// TIA Portal project "Hydaulikaggregat" (V14)

(* hardware
DEVICE "S7-1200-Station_1"  S7-1200 Station
   slot 0: "Baugruppenträger_0"  Rack  V1.0
   slot 1: "PLC"  CPU 1214C DC/DC/DC  6ES7 214-1AG40-0XB0  V4.1
   slot 3: "AQ 1x12BIT_1"  6ES7 232-4HA30-0XB0  V1.0
DEVICE "HMI"  KTP700 Basic PN
   slot 0: "HMI"  HMI  6AV2 123-2GB03-0AX0  13.0.1.0
   slot 1: "HMI_RT_1"  KTP700 Basic PN  6AV2 123-2GB03-0AX0  13.0.1.0
   slot 5: "HMI.IE_CP_1"  PROFINET Schnittstelle
      slot 1: "PROFINET Schnittstelle_1"  PROFINET Schnittstelle
         slot 1: "Port_1"  Port
*)

// ===== PLC "PLC"  CPU 1214C DC/DC/DC =====

VAR_GLOBAL   // PLC tag table "Standard-Variablentabelle"
   "System_Byte" AT %MB100 : Byte;
   "FirstScan" AT %M100.0 : Bool;
   "DiagStatusUpdate" AT %M100.1 : Bool;
   "AlwaysTRUE" AT %M100.2 : Bool;
   "AlwaysFALSE" AT %M100.3 : Bool;
   "Clock_Byte" AT %MB110 : Byte;
   "Clock_10Hz" AT %M110.0 : Bool;
   "Clock_5Hz" AT %M110.1 : Bool;
   "Clock_2.5Hz" AT %M110.2 : Bool;
   "Clock_2Hz" AT %M110.3 : Bool;
   "Clock_1.25Hz" AT %M110.4 : Bool;
   "Clock_1Hz" AT %M110.5 : Bool;
   "Clock_0.625Hz" AT %M110.6 : Bool;
   "Clock_0.5Hz" AT %M110.7 : Bool;
   "S1 Taster Start" AT %Q0.0 : Bool;
   "S2 Taster Stop" AT %Q0.1 : Bool;
   "S3 Taster Quittieren" AT %Q0.2 : Bool;
   "B1Füllstand Ölbehälter" AT %Q0.3 : Bool;
   "B2 Öl Druck erreicht" AT %Q0.4 : Bool;
   "B3 Öl Überdruck" AT %Q0.5 : Bool;
   "F5 Motorschutzschalter" AT %Q0.6 : Bool;
   "Q1 Netzschütz" AT %I0.0 : Bool;
   "Q2 Sternschütz" AT %I0.1 : Bool;
   "Q3 Dreieckschütz" AT %I0.2 : Bool;
   "P1 Störung Motor" AT %I0.3 : Bool;
   "P2 Überdruck" AT %I0.4 : Bool;
   "P3 Druck erreicht" AT %I0.5 : Bool;
   "P4 Ölstand min." AT %I0.6 : Bool;
   "ÖlPegel" AT %MW20 : Int;
   "ÖlPegelReal" AT %MD22 : Real;
   "ÖlDruck" AT %MW26 : Int;
   "ÖlDruckReal" AT %MD28 : Real;
   "Knopf Öl nachfüllen" AT %M10.0 : Bool;
   "Impulsmerker_100ms" AT %M10.1 : Bool;
   "Q1 Netzschütz alt" AT %M10.2 : Bool;
   "Betriebsart" AT %MW40 : Int;
   "Pegelrechner" AT %MW42 : Int;
   "ÖlpegelAnzeige" AT %MW44 : Int;
   "Text Normalbetrieb" AT %M10.5 : Bool;
   "Text Druckproblem" AT %M10.6 : Bool;
   "Text Ölpegelproblem" AT %M10.7 : Bool;
   "AlleAusgänge" AT %QW0 : Word;
END_VAR

// folder: System blocks/Program resources

DATA_BLOCK "Impulsgeber_100ms"   // DB2
{ S7_Optimized_Access := 'TRUE' }
AUTHOR : Simatic
FAMILY : IEC
NAME : IEC_TMR
VERSION : 1.0
// stored: InstanceOfName IEC_TIMER
"IEC_TIMER"
BEGIN
END_DATA_BLOCK

// folder: (top level)

FUNCTION "fc_Hydraulikaggregat" : Void   // FC1, SCL
{ S7_Optimized_Access := 'TRUE' }
VERSION : 0.1
BEGIN
   "Impulsgeber_100ms".TON(IN:=NOT "Impulsmerker_100ms",
                           PT:=t#100ms,
                           Q=>"Impulsmerker_100ms"
   );

   IF "Knopf Öl nachfüllen" THEN
       "ÖlPegelReal" := 1000;
       "Pegelrechner" := 0;
   END_IF;

   // Es gibt drei Betriebsarten; sie werden immer beim Starten des Motors umgeschaltet
   // 1 ... Normalbetrieb: Pegel bleibt voll; Druck steigt bis 70%
   // 0 ... Es sinkt der Pegel nach und nach ab
   // 2 ... Es steigt der Betriebsdruck an

   IF "Q1 Netzschütz" AND NOT "Q1 Netzschütz alt" THEN
       "Betriebsart" := "Betriebsart" + 1;
   END_IF;
   "Q1 Netzschütz alt" := "Q1 Netzschütz";

   CASE "Betriebsart" OF
       0:
           "Text Normalbetrieb" := FALSE;
           "Text Ölpegelproblem" := TRUE;
           "Text Druckproblem" := FALSE;
       1:
           "Text Normalbetrieb" := TRUE;
           "Text Ölpegelproblem" := FALSE;
           "Text Druckproblem" := FALSE;
       2:
           "Text Normalbetrieb" := FALSE;
           "Text Ölpegelproblem" := FALSE;
           "Text Druckproblem" := TRUE;
       ELSE
           "Betriebsart" := 0;
   END_CASE;


   IF "Impulsmerker_100ms" THEN

       IF "ÖlDruckReal" > 0 AND NOT "Q1 Netzschütz" THEN
           "ÖlDruckReal" := "ÖlDruckReal" - 20;            // Motor AUS --> Druck sinkt rapide
       END_IF;

       IF "Q1 Netzschütz" AND "Q2 Sternschütz" THEN
           "ÖlDruckReal" := "ÖlDruckReal" + 2;             // Motor Stern --> Druck steigt langsam
       END_IF;

       IF "Q1 Netzschütz" AND "Q3 Dreieckschütz" THEN
           "ÖlDruckReal" := "ÖlDruckReal" + 10;            // Motor Dreieck --> Druck steigt schneller
       END_IF;


       CASE "Betriebsart" OF
           1:  // Normalbetrieb; nach dem ersten Mal Motor EIN
               "Pegelrechner" := 0;
               "ÖlPegelReal" := 1000;
               IF "ÖlDruckReal" > 700 THEN
                   "ÖlDruckReal" := 700;
               END_IF;
           2:  // Es kommt zu Überdruck
               "Pegelrechner" := 0;
               "ÖlPegelReal" := 1000;
               IF "ÖlDruckReal" > 900 THEN
                   "ÖlDruckReal" := 900;
               END_IF;
           0:  // Ölpegel schwank 
               IF "ÖlDruckReal" > 700 THEN
                   "ÖlDruckReal" := 700;
               END_IF;

               IF "Pegelrechner" < 1000 THEN
                   "Pegelrechner" := "Pegelrechner" + 2;
               ELSE
                   "Pegelrechner" := 0;
               END_IF;

               CASE "Pegelrechner" OF
                   0..100:     "ÖlPegelReal" := "ÖlPegelReal" - 2;
                   100..150:   "ÖlPegelReal" := "ÖlPegelReal" + 1;
                   150..250:   "ÖlPegelReal" := "ÖlPegelReal" - 2;
                   250..300:   "ÖlPegelReal" := "ÖlPegelReal" + 1;
                   300..400:   "ÖlPegelReal" := "ÖlPegelReal" - 2;
                   400..450:   "ÖlPegelReal" := "ÖlPegelReal" + 1;
                   450..550:   "ÖlPegelReal" := "ÖlPegelReal" - 2;
                   550..600:   "ÖlPegelReal" := "ÖlPegelReal" + 1;
                   600..700:   "ÖlPegelReal" := "ÖlPegelReal" - 2;
                   700..750:   "ÖlPegelReal" := "ÖlPegelReal" + 1;
                   750..850:   "ÖlPegelReal" := "ÖlPegelReal" - 2;
                   850..900:   "ÖlPegelReal" := "ÖlPegelReal" + 1;
               END_CASE;
       END_CASE;
   END_IF;

   IF "ÖlDruckReal" > 1000 THEN
       "ÖlDruckReal" := 0;
   END_IF;

   IF "ÖlDruckReal" > 600 THEN
       "B2 Öl Druck erreicht" := TRUE;
   ELSE
       "B2 Öl Druck erreicht" := FALSE;
   END_IF;

   IF "ÖlDruckReal" > 800 THEN
       "B3 Öl Überdruck" := TRUE;
   ELSE
       "B3 Öl Überdruck" := FALSE;
   END_IF;

   IF "ÖlPegelReal" > 250 THEN          
       "B1Füllstand Ölbehälter" := true;
   ELSE
       "B1Füllstand Ölbehälter" := FALSE;
   END_IF;

   IF "ÖlDruckReal" < 0 THEN
       "ÖlDruckReal" := 0;
   END_IF;

   IF "ÖlPegelReal" < 0 THEN
       "ÖlPegelReal" := 0;
   END_IF;

   "ÖlDruck" := "ÖlDruckReal" / 10;        // Promille in % umrechnen
   "ÖlpegelAnzeige" := "ÖlPegelReal" / 10; // Promille in % umrechnen 
   "ÖlPegel" := 100 - "ÖlpegelAnzeige";
END_FUNCTION

ORGANIZATION_BLOCK "Main"   // OB1, LAD, ProgramCycle
TITLE = "Main Program Sweep (Cycle)"
{ S7_Optimized_Access := 'TRUE' }
VERSION : 0.1
   VAR_INPUT
      Initial_Call : Bool;   // Initial call of this OB
      Remanence : Bool;   // =True, if remanent data are available
   END_VAR
BEGIN

REGION Network 1: -Q1
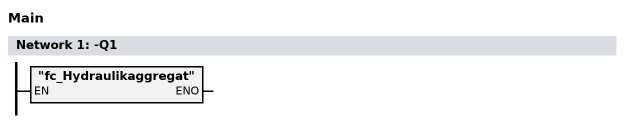
   RUNG wire#powerrail
      "fc_Hydraulikaggregat"()
   END_RUNG
   // the same network as SCL:
   "fc_Hydraulikaggregat"();
END_REGION
END_ORGANIZATION_BLOCK

ORGANIZATION_BLOCK "Startup"   // OB100, SCL, Startup
TITLE = "Complete Restart"
{ S7_Optimized_Access := 'TRUE' }
VERSION : 0.1
   VAR_INPUT
      LostRetentive : Bool;   // True if retentive data are lost
      LostRTC : Bool;   // True if date and time are lost
   END_VAR
BEGIN
   "AlleAusgänge" := 16#0000;
END_ORGANIZATION_BLOCK

(* ===== HMI "HMI_RT_1" =====
system functions are stored by id; their names below are inferred from use
connection "HMI_Verbindung_1": ETHERNET, SMART_S7_1200_OMS

HMI tags "Standard-Variablentabelle"
   "AlwaysTRUE" : Bool = PLC AlwaysTRUE AT %M100.2, 100 ms
   "P1 Störung Motor" : Bool = PLC "P1 Störung Motor" AT %I0.3, 100 ms
   "P2 Überdruck" : Bool = PLC "P2 Überdruck" AT %I0.4, 100 ms
   "P3 Druck erreicht" : Bool = PLC "P3 Druck erreicht" AT %I0.5, 100 ms
   "P4 Ölstand min." : Bool = PLC "P4 Ölstand min." AT %I0.6, 100 ms
   "Knopf Öl nachfüllen" : Bool = PLC "Knopf Öl nachfüllen" AT %M10.0, 100 ms
   "F5 Motorschutzschalter" : Bool = PLC "F5 Motorschutzschalter" AT %Q0.6, 100 ms
   "S1 Taster Start" : Bool = PLC "S1 Taster Start" AT %Q0.0, 100 ms
   "S2 Taster Stop" : Bool = PLC "S2 Taster Stop" AT %Q0.1, 100 ms
   "S3 Taster Quittieren" : Bool = PLC "S3 Taster Quittieren" AT %Q0.2, 100 ms
   "Q1 Netzschütz" : Bool = PLC "Q1 Netzschütz" AT %I0.0, 100 ms
   "Q2 Sternschütz" : Bool = PLC "Q2 Sternschütz" AT %I0.1, 100 ms
   "Q3 Dreieckschütz" : Bool = PLC "Q3 Dreieckschütz" AT %I0.2, 100 ms
   "B1Füllstand Ölbehälter" : Bool = PLC "B1Füllstand Ölbehälter" AT %Q0.3, 100 ms
   "B2 Öl Druck erreicht" : Bool = PLC "B2 Öl Druck erreicht" AT %Q0.4, 100 ms
   "B3 Öl Überdruck" : Bool = PLC "B3 Öl Überdruck" AT %Q0.5, 100 ms
   "ÖlDruck" : Int = PLC ÖlDruck AT %MW26, 100 ms
   "ÖlPegel" : Int = PLC ÖlPegel AT %MW20, 100 ms
   "ÖlpegelAnzeige" : Int = PLC ÖlpegelAnzeige AT %MW44, 100 ms
   "Text Normalbetrieb" : Bool = PLC "Text Normalbetrieb" AT %M10.5, 100 ms
   "Text Druckproblem" : Bool = PLC "Text Druckproblem" AT %M10.6, 100 ms
   "Text Ölpegelproblem" : Bool = PLC "Text Ölpegelproblem" AT %M10.7, 100 ms

screen "Hydraulikaggregat" 800x480
   TextField "Textfeld_2" at 197,4 size 528x43; Text 'Hydraulikaggregat - Digital Twin'
   Button "Schaltfläche_1" at 615,65 size 80x40; TextOff 'Start'
      on Press: SetBit("S1 Taster Start")
      on Release: ResetBit("S1 Taster Start")
   Button "Schaltfläche_2" at 702,65 size 80x40; TextOn 'Automatik'; TextOff 'Stop'
      on Release: SetBit("S2 Taster Stop")
      on Press: ResetBit("S2 Taster Stop")
   Button "Schaltfläche_4" at 615,420 size 170x50; TextOn 'Thermo 1'; TextOff 'Motorschutz'
      on Click: InvertBit("F5 Motorschutzschalter")
      Appearance <- "F5 Motorschutzschalter"
   Circle "Kreis_3" at 610,210 size 50x50
      Appearance <- "P2 Überdruck"
   TextField "Textfeld_4" at 660,225 size 89x23; Text 'Überdruck'
   Circle "Kreis_5" at 610,160 size 50x50
      Appearance <- "P1 Störung Motor"
   TextField "Textfeld_6" at 660,175 size 127x23; Text 'Störung Motor'
   Button "Schaltfläche_3" at 612,110 size 170x40; TextOn 'Automatik'; TextOff 'Quittieren'
      on Release: ResetBit("S3 Taster Quittieren")
      on Press: SetBit("S3 Taster Quittieren")
   Circle "Kreis_1" at 610,260 size 50x50
      Appearance <- "P3 Druck erreicht"
   Circle "Kreis_2" at 610,310 size 50x50
      Appearance <- "P4 Ölstand min."
   TextField "Textfeld_1" at 660,275 size 121x23; Text 'Druck erreicht'
   TextField "Textfeld_3" at 660,325 size 107x23; Text 'Ölstand min.'
   GraphicView "Grafikanzeige_1" at 379,300 size 30x30; Picture "HMI_Symbole_Schwimmerschalter_Schliesser"
      Visibility <- "F5 Motorschutzschalter"
   GraphicView "Grafikanzeige_2" at 376,300 size 40x30; Picture "HMI_Symbole_Schwimmerschalter_Schliesser_Betaetigt"
      Visibility <- "F5 Motorschutzschalter"
   GraphicView "Grafikanzeige_3" at 471,300 size 30x30; Picture "HMI_Symbole_Schwimmerschalter_Schliesser"
      Visibility <- "B2 Öl Druck erreicht"
   GraphicView "Grafikanzeige_4" at 466,300 size 40x30; Picture "HMI_Symbole_Schwimmerschalter_Schliesser_Betaetigt"
      Visibility <- "B2 Öl Druck erreicht"
   GraphicView "Grafikanzeige_5" at 516,300 size 30x30; Picture "HMI_Symbole_Schwimmerschalter_Schliesser"
      Visibility <- "B3 Öl Überdruck"
   GraphicView "Grafikanzeige_6" at 511,300 size 40x30; Picture "HMI_Symbole_Schwimmerschalter_Schliesser_Betaetigt"
      Visibility <- "B3 Öl Überdruck"
   TextField "Textfeld_5" at 380,281 size 24x23; Text 'F5'
   TextField "Textfeld_7" at 475,281 size 26x23; Text 'B2'
   TextField "Textfeld_8" at 516,281 size 26x23; Text 'B3'
   GraphicView "Grafikanzeige_7" at 26,380 size 40x30; Picture "HMI_Symbole_Schwimmerschalter_Schliesser_Betaetigt"
      Visibility <- "B1Füllstand Ölbehälter"
   GraphicView "Grafikanzeige_8" at 30,380 size 30x30; Picture "HMI_Symbole_Schwimmerschalter_Schliesser"
      Visibility <- "B1Füllstand Ölbehälter"
   TextField "Textfeld_9" at 26,357 size 26x23; Text 'B1'
   TextField "Textfeld_10" at 367,368 size 29x23; Text 'M1'
   Rectangle "Rechteck_5" at 346,342 size 35x25
      Appearance <- "Q2 Sternschütz"
   TextField "Textfeld_11" at 357,342 size 16x23; Text 'Y'
   Rectangle "Rechteck_6" at 380,342 size 35x25
      Appearance <- "Q3 Dreieckschütz"
   TextField "Textfeld_12" at 389,342 size 17x23; Text 'D'
   Bar "Balken_1" at 445,64 size 135x219; MinimumValue 0; MaximumValue 100
      ProcessValue <- "ÖlDruck"
   Rectangle "Rechteck_9" at 76,91 size 241x168
      VerticalMovement <- "ÖlPegel"
   Button "Schaltfläche_6" at 82,130 size 93x52; TextOff 'Nachfüllen'
      on Press: SetBit("Knopf Öl nachfüllen")
      on Release: ResetBit("Knopf Öl nachfüllen")
   Circle "Kreis_4" at 348,387 size 64x64
      Appearance <- "Q1 Netzschütz"
   IOField "EA-Feld_1" at 144,391 size 96x32; FormatPattern s99999
      ProcessValue <- "ÖlpegelAnzeige"
   TextField "Textfeld_13" at 15,70 size 123x23; Text 'Normalbetrieb'
      Visibility <- "Text Normalbetrieb"
   TextField "Textfeld_14" at 15,70 size 182x23; Text 'Probleme mit Öldruck'
      Visibility <- "Text Druckproblem"
   TextField "Textfeld_15" at 15,70 size 366x23; Text 'Probleme mit dem Füllstand des Ölbehälters'
      Visibility <- "Text Ölpegelproblem"
*)